// TIA Portal V16 export
// export: Created 2024-09-05T17:40:13.5402899Z, ExportSetting WithDefaults, DisplayName Totally Integrated Automation Portal, DisplayVersion V16 Update 6, DisplayName TIA Portal Version Control Interface, DisplayVersion V16 Update 2, DisplayName TIA Portal Openness, DisplayVersion V16 Update 6, DisplayName STEP 7 Professional, DisplayVersion V16 Update 6, DisplayName STEP 7 Safety, DisplayVersion V16, DisplayName WinCC Advanced, DisplayVersion V16 Update 6
TYPE "UDT_EksKey"
// stored: IsFailsafeCompliant false
   STRUCT
      Level : Int;
      EmployeeID : Array[1..4] of Char;
      KeyID : Array[1..16] of Char;
      Comment : Array[1..20] of Char;
   END_STRUCT;
END_TYPE
